# EPICS autosave request: iocBoot/ioc13lab_tomoCollect/auto_settings.req
file "TomoCollect_settings.req",        P=$(P), R=TC:
